{attribute 'OPC.UA.DA.StructuredType' := '1'}
TYPE ST_StrategySetParameters :
STRUCT
	bProductionModeActivated : BOOL; //true if thermal networks should be controlled according to production mode
END_STRUCT
END_TYPE

(* stored: Version 1.1.0.1, ProductVersion 3.1.4024.10
   DUT ST_StrategySetParameters: Id {bf7c7f5f-b067-4346-9be2-2c3102008760} *)
